// LS Electric XG5000 project: Timer
// PLC LSPLC

PROGRAM NewProgram2 (task: 스캔 프로그램)

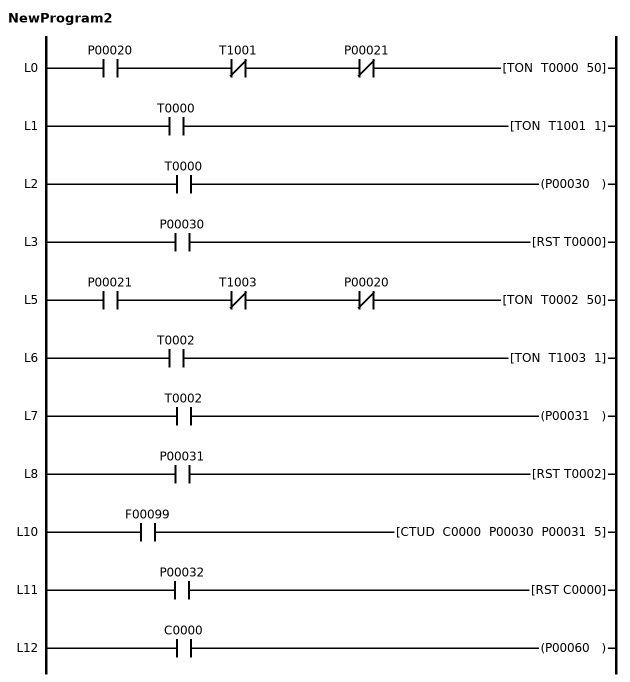
; L0
LOAD      P00020
AND NOT   T1001
AND NOT   P00021
TON       T0000 50
; L1
LOAD      T0000
TON       T1001 1
; L2
LOAD      T0000
OUT       P00030
; L3
LOAD      P00030
RST       T0000
; L5
LOAD      P00021
AND NOT   T1003
AND NOT   P00020
TON       T0002 50
; L6
LOAD      T0002
TON       T1003 1
; L7
LOAD      T0002
OUT       P00031
; L8
LOAD      P00031
RST       T0002
; L10
LOAD      F00099
CTUD      C0000 P00030 P00031 5
; L11
LOAD      P00032
RST       C0000
; L12
LOAD      C0000
OUT       P00060